// TIA Portal V20 export
FUNCTION_BLOCK "FB_BwControl"   // FB39, SCL
{ S7_Optimized_Access := 'TRUE' }
// stored: MemoryReserve 100, SetENOAutomatically false
   VAR_INPUT
      iStartSeqCond : Bool;   // Start Sequence Conditions
      iJobReq : Bool;   // Job Request - From Main
      iCtrlEnabled : Bool;   // Part Control Enable - Param or Condition
      iShuttleCtrlPos : Bool;   // Control Pos. Reached - Param
      iShuttleCtrlPosSetPoint : LReal;   // Control Pos. Setpoint - Param
      iExpectedCtrl : Bool;   // Expected result ctrl
      iBwPresence : Bool;   // Bw Presence - From DI
      iShuttleMoving : Bool;   // Shuttle is moving - From FB_LoaderAxis
      iShuttleInPos : Bool;   // Shuttle pos. reached - From FB_LoaderAxis
      iPLC_DateAndTime : DTL;
      iStepPause : Bool;
   END_VAR
   VAR_OUTPUT
      oShuttleStartReq { ExternalAccessible := 'False'; ExternalVisible := 'False'; ExternalWritable := 'False'} : Bool;   // Shuttle Start Order - To FB_LoaderAxis
      oShuttlePosSetPoint { ExternalAccessible := 'False'; ExternalVisible := 'False'; ExternalWritable := 'False'} : Real;   // Shuttle Position Setpoint - To FB_LoaderAxis
      oBwControlOK : Bool;   // Bw OK - To Main
      oBwControlNOK : Bool;   // Bw NOK - To Main
   END_VAR
   VAR
      sCurrent_Step_NB : Int;   // Active Step Number
      sCheck_Step_Condition : Bool;
      sOneStepForward : Bool;
      sRTOneStepForward : R_TRIG;
      sOneStepMode { S7_SetPoint := 'True'} : Bool;
      sStepForward : Bool;
      sInterface : "UDT_SequenceInterface";
      sShuttleStartReq { ExternalAccessible := 'False'; ExternalVisible := 'False'; ExternalWritable := 'False'} : Bool;
      sShuttlePosSetPoint { ExternalAccessible := 'False'; ExternalVisible := 'False'; ExternalWritable := 'False'} : Real;
      sMissingBwCtrl : Bool;
      sExtraBwCtrl : Bool;
      sPresenceBw : Bool;
      sBwControlOK : Bool;
      sBwControlNOK : Bool;
      sHistory : Struct
         Activation : Bool;
         Steps : Array[0..99] of Int;
         Date_Time : Array[0..99] of DTL;
      END_STRUCT;
      StepText : "FB_GetTextErrorCode";
   END_VAR
   VAR_TEMP
      tIndex : Int;   // Index
   END_VAR
   VAR CONSTANT
      S00_INIT : Int := 0;
      S10_CHECK_BW_PRESENCE_OPTION : Int := 10;
      S20_SHUTTLE_TO_BW_CTRL_POS_START_REQ : Int := 20;
      S30_SHUTTLE_TO_BW_CTRL_POS_REACHED : Int := 30;
      S40_WAIT_BW_CTRL_EXECUTION : Int := 40;
      S50_CHECK_BW_PRES_RESULT : Int := 50;
      S150_SET_BW_PRES_RESULT : Int := 150;
      S195_JOB_DONE : Int := 195;
   END_VAR
   // StepText.sCode_error[0].ErrorCode := 0;
   // StepText.sCode_error[1].ErrorCode := 10;
   // StepText.sCode_error[2].ErrorCode := 20;
   // StepText.sCode_error[3].ErrorCode := 30;
   // StepText.sCode_error[4].ErrorCode := 40;
   // StepText.sCode_error[5].ErrorCode := 50;
   // StepText.sCode_error[6].ErrorCode := 60;
   // StepText.sCode_error[7].ErrorCode := 70;
   // StepText.sCode_error[8].ErrorCode := 80;
   // StepText.sCode_error[9].ErrorCode := 90;
   // StepText.sCode_error[10].ErrorCode := 95;
BEGIN
   REGION Description header 
       //==================================================================================
       // POSALUX Swiss SA / (C) Copyright 2025
       //----------------------------------------------------------------------------------
       // Title: FB_BwControl
       // Comment/Function: 
       // Author: Fabien WALDT
       // Engineering: TIA Portal v17
       //----------------------------------------------------------------------------------
       // Change log table:
       // Version  | Date     | Expert in charge | Changes applied
       // ---------|----------|------------------|-----------------------------------------
       // 00.00.01 | 20250527 | WFA              | First released version
       // =================================================================================
   END_REGION

   REGION Define condition to start
       IF #iStartSeqCond THEN
           #sInterface.SequenceReleased := TRUE;
       ELSE
           // Standard sequencer controls
           #sInterface.SequenceReleased := FALSE;
           #sCurrent_Step_NB := #S00_INIT;
           #sInterface.SequenceRun := FALSE;
           #sInterface.JobDone := FALSE;
           #sCheck_Step_Condition := FALSE;

           // Dedicated sequencer controls
           #sShuttleStartReq := FALSE;
           #sShuttlePosSetPoint := 0.0;
           #sPresenceBw := FALSE;

           // Add specifics controls 
       END_IF;

       // Reset interface error
       IF #sInterface.Reset THEN
           #sInterface.Error := FALSE;
       END_IF;

       // Reset start when axis in position
       IF #iShuttleInPos THEN
           #sShuttleStartReq := FALSE;
       END_IF;

       // One step forward
       #sRTOneStepForward.CLK := #sOneStepForward;
       #sRTOneStepForward();
       #sStepForward := (NOT #sOneStepMode OR (#sOneStepMode AND #sRTOneStepForward.Q)) AND NOT #iStepPause;
       #sOneStepForward := FALSE;
   END_REGION

   REGION Sequence Function
       CASE #sCurrent_Step_NB OF
           #S00_INIT:
               REGION S00 INIT
                   #sCheck_Step_Condition := TRUE;
               END_REGION
           #S10_CHECK_BW_PRESENCE_OPTION:
               REGION S10_CHECK_BW_PRESENCE_OPTION
                   #sBwControlOK := FALSE;
                   #sBwControlNOK := FALSE;
                   #sMissingBwCtrl := FALSE;
                   #sExtraBwCtrl := FALSE;
                   #sCheck_Step_Condition := TRUE;
               END_REGION
           #S20_SHUTTLE_TO_BW_CTRL_POS_START_REQ:
               REGION S20_SHUTTLE_TO_BW_CTRL_POS_START_REQ
                   #sShuttleStartReq := NOT #iShuttleCtrlPos;
                   #sShuttlePosSetPoint := LREAL_TO_REAL(#iShuttleCtrlPosSetPoint);
                   #sCheck_Step_Condition := TRUE;
               END_REGION
           #S30_SHUTTLE_TO_BW_CTRL_POS_REACHED:
               REGION S30_SHUTTLE_TO_BW_CTRL_POS_REACHED
                   #sCheck_Step_Condition := TRUE;
               END_REGION
           #S40_WAIT_BW_CTRL_EXECUTION:
               REGION S40_WAIT_BW_CTRL_EXECUTION
                   #sPresenceBw := #iBwPresence;
                   #sCheck_Step_Condition := TRUE;
               END_REGION
           #S50_CHECK_BW_PRES_RESULT:
               REGION S50_CHECK_BW_PRES_RESULT
                   #sExtraBwCtrl := #sPresenceBw AND NOT #iExpectedCtrl;
                   #sMissingBwCtrl := NOT #sPresenceBw AND #iExpectedCtrl;
                   IF #sPresenceBw = #iExpectedCtrl THEN
                       #sBwControlOK := TRUE;
                       #sBwControlNOK := FALSE;
                   ELSE
                       #sBwControlOK := FALSE;
                       #sBwControlNOK := TRUE;
                   END_IF;
                   #sCheck_Step_Condition := TRUE;
               END_REGION
           #S150_SET_BW_PRES_RESULT:
               REGION S150_SET_BW_PRES_RESULT
                   #sBwControlOK := TRUE;
                   #sBwControlNOK := FALSE;
                   #sCheck_Step_Condition := TRUE;
               END_REGION
           #S195_JOB_DONE:
               REGION S195_JOB_DONE
                   #sInterface.JobDone := TRUE;
                   #sCheck_Step_Condition := TRUE;
               END_REGION
           ELSE:
               #sInterface.Error := TRUE;
       END_CASE;
   END_REGION

   REGION Sequence Next Step Condition
       IF #sCheck_Step_Condition THEN
           CASE #sCurrent_Step_NB OF
               #S00_INIT:
                   REGION S00 INIT
                       IF #sInterface.SequenceReleased AND #iJobReq THEN
                           #sCurrent_Step_NB := #S10_CHECK_BW_PRESENCE_OPTION;
                           #sInterface.SequenceRun := TRUE;
                           #sCheck_Step_Condition := FALSE;
                       ELSE
                           #sInterface.SequenceRun := FALSE;
                       END_IF;
                   END_REGION
               #S10_CHECK_BW_PRESENCE_OPTION:
                   REGION S10_CHECK_BW_PRESENCE_OPTION
                       IF #sInterface.SequenceReleased AND #sStepForward AND "DB_LoaderOptions".BwControl.UndrilledDrilledCtrlSeparate AND (NOT "DB_LoaderOptions".BwControl.Disabled OR NOT #iCtrlEnabled) THEN
                           #sCurrent_Step_NB := #S20_SHUTTLE_TO_BW_CTRL_POS_START_REQ;
                           #sCheck_Step_Condition := FALSE;
                       ELSIF #sInterface.SequenceReleased AND #sStepForward AND ("DB_LoaderOptions".BwControl.Disabled OR NOT #iCtrlEnabled) THEN
                           #sCurrent_Step_NB := #S150_SET_BW_PRES_RESULT;
                           #sCheck_Step_Condition := FALSE;
                       END_IF;
                   END_REGION
               #S20_SHUTTLE_TO_BW_CTRL_POS_START_REQ:
                   REGION S20_SHUTTLE_TO_BW_CTRL_POS_START_REQ
                       IF #sInterface.SequenceReleased AND (#iShuttleMoving OR #iShuttleCtrlPos) THEN
                           #sCurrent_Step_NB := #S30_SHUTTLE_TO_BW_CTRL_POS_REACHED;
                           #sCheck_Step_Condition := FALSE;
                       END_IF;
                   END_REGION
               #S30_SHUTTLE_TO_BW_CTRL_POS_REACHED:
                   REGION S30_SHUTTLE_TO_BW_CTRL_POS_REACHED
                       IF #sInterface.SequenceReleased AND #sStepForward AND NOT #sShuttleStartReq AND #iShuttleCtrlPos THEN
                           #sCurrent_Step_NB := #S40_WAIT_BW_CTRL_EXECUTION;
                           #sCheck_Step_Condition := FALSE;
                       END_IF;
                   END_REGION
               #S40_WAIT_BW_CTRL_EXECUTION:
                   REGION S40_WAIT_BW_CTRL_EXECUTION
                       IF #sInterface.SequenceReleased AND #sStepForward AND "AlwaysTRUE" THEN
                           #sCurrent_Step_NB := #S50_CHECK_BW_PRES_RESULT;
                           #sCheck_Step_Condition := FALSE;
                       END_IF;
                   END_REGION
               #S50_CHECK_BW_PRES_RESULT:
                   REGION S50_CHECK_BW_PRES_RESULT
                       IF #sInterface.SequenceReleased AND #sStepForward AND "AlwaysTRUE" THEN
                           #sCurrent_Step_NB := #S195_JOB_DONE;
                           #sCheck_Step_Condition := FALSE;
                       END_IF;
                   END_REGION
               #S150_SET_BW_PRES_RESULT:
                   REGION S150_SET_BW_PRES_RESULT
                       IF #sInterface.SequenceReleased AND #sStepForward AND "AlwaysTRUE" THEN
                           #sCurrent_Step_NB := #S195_JOB_DONE;
                           #sCheck_Step_Condition := FALSE;
                       END_IF;
                   END_REGION
               #S195_JOB_DONE:
                   REGION S195_JOB_DONE
                       IF NOT #iJobReq THEN
                           #sCurrent_Step_NB := #S00_INIT;
                           #sCheck_Step_Condition := FALSE;
                           #sInterface.JobDone := FALSE;
                       END_IF;
                   END_REGION
               ELSE
                   #sInterface.Error := TRUE;
           END_CASE;
       END_IF;
   END_REGION

   REGION Outputs Update
       #oShuttleStartReq := #sShuttleStartReq;
       #oShuttlePosSetPoint := #sShuttlePosSetPoint;
       #oBwControlOK := #sBwControlOK;
       #oBwControlNOK := #sBwControlNOK;
   END_REGION

   REGION Steps - Date and Time History
       IF #sHistory.Activation THEN
           IF #sHistory.Steps[0] <> #sCurrent_Step_NB THEN
               FOR #tIndex := 98 TO 0 BY -1 DO
                   #sHistory.Steps[#tIndex + 1] := #sHistory.Steps[#tIndex];
                   #sHistory.Date_Time[#tIndex + 1] := #sHistory.Date_Time[#tIndex];
               END_FOR;
               #sHistory.Steps[0] := #sCurrent_Step_NB;
               #sHistory.Date_Time[0] := #iPLC_DateAndTime;
           END_IF;
       END_IF;
   END_REGION

   REGION Steps Text
       #StepText(iErrorCode := #sCurrent_Step_NB,
                 oErrorText => #StepText.oErrorText);
   END_REGION
END_FUNCTION_BLOCK
